FUNCTION_BLOCK FB_InAnotherTouch
VAR_INPUT
	CurrTouchIdx	: INT;
	CurrentIdx		: DINT;
	TouchConfig		: ARRAY [1..TouchNo] OF ST_TouchConfig;
	TouchConfigIdx	: ARRAY [1..TouchNo] OF  INT;
END_VAR
VAR_OUTPUT
	Yes				:BOOL;
END_VAR
VAR
	touchIdx			:INT;
END_VAR


Yes := FALSE;

FOR touchIdx := 1 TO TouchNo DO
	IF touchIdx <> CurrTouchIdx
	AND CurrentIdx > TouchConfig[touchIdx].StartIdx[TouchConfigIdx[touchIdx]]
	AND CurrentIdx < TouchConfig[touchIdx].EndIdx[TouchConfigIdx[touchIdx]] THEN
		Yes := TRUE;
	END_IF
END_FOR

END_FUNCTION_BLOCK

(* stored: Version 1.1.0.1, ProductVersion 3.1.4024.9
   POU FB_InAnotherTouch: Id {0579c938-78b7-4194-8a37-943e7d1744e4}, SpecialFunc None *)
